{attribute addProperty BoxType "EL3208-0000-0017"}
{attribute addProperty Id "RTD_Inputs_ChannelAT %I*ARRAY[0..7] OF RTD_Inputs_Channel_17AE08DB256320WcStateAT %I*WcState_F855686C1620InfoDataAT %I*InfoData_BC63D37F80100"}
{attribute addProperty CRC "9594934"}
{attribute addProperty SizeInBites "352"}
{attribute addProperty SizeInBytes "44"}
TYPE EL3208_6C7FE116 :
STRUCT
	{attribute addProperty Name "RTD_Inputs_Channel"}
	RTD_Inputs_Channel : ARRAY[0..7] OF RTD_Inputs_Channel_17AE08DB;
	{attribute addProperty Name "WcState"}
	WcState : WcState_F855686C;
	{attribute addProperty Name "InfoData"}
	InfoData : InfoData_BC63D37F;
END_STRUCT
END_TYPE

(* stored: Version 1.2.0.0, ProductVersion 3.1.4024.9
   DUT EL3208_6C7FE116: Id {36102ef1-7257-4558-a996-3404fa97a82c} *)
